// TIA Portal V19 export
VAR_GLOBAL   // PLC tag table "D24"
   D24_Lp_EntryReq_LB307 AT %Q300.2 : Bool;   // 270SH1
   D24_Lp_EntryReq_LB308 AT %Q350.2 : Bool;   // 271SH1
   D24_Lp_SafetyReset_LB307 AT %Q300.3 : Bool;   // 270SH2
   D24_Lp_SafetyReset_LB308 AT %Q350.3 : Bool;   // 271SH2
   D24_Pb_EntryReq_LB307 AT %I300.5 : Bool;   // 270SH1
   D24_Pb_EntryReq_LB308 AT %I350.2 : Bool;   // 271SH1
   D24_Pb_SafetyReset_LB307 AT %I300.6 : Bool;   // 270SH2
   D24_Pb_SafetyReset_LB308 AT %I350.3 : Bool;   // 271SH2
   D24_Ls AT %I1400.3 : Bool;   // 300DI3 - 270BE1/R1
END_VAR
